// TIA Portal project "2022.11.22_双轴仿真2" (V17)
// Vorlageprojekt für das Buch mit Zielsystem S7-1200

(* hardware
DEVICE "S7-1200-Station_1"  S7-1200 Station
   slot 0: "Baugruppenträger_0"  Rack  V1.0
   slot 1: "PLC_1"  CPU 1214C DC/DC/DC  6ES7 214-1AG40-0XB0  V4.5
*)

// ===== PLC "PLC_1"  CPU 1214C DC/DC/DC =====

VAR_GLOBAL   // PLC tag table "Standard-Variablentabelle"
   "感应器5" AT %I1.1 : Bool;
   "感应器6" AT %I1.2 : Bool;
   "输入预留3" AT %I1.3 : Bool;
   "输入预留4" AT %I1.4 : Bool;
   "输入预留5" AT %I1.5 : Bool;
   "输入预留6" AT %I1.6 : Bool;
   "输入预留7" AT %I1.7 : Bool;
   "传送带4" AT %Q0.3 : Bool;
   "输出预留2" AT %Q0.7 : Bool;
   "输出预留3" AT %Q1.2 : Bool;
   "输出预留4" AT %Q1.5 : Bool;
   "输出预留5" AT %Q1.6 : Bool;
   "输出预留6" AT %Q1.7 : Bool;
   "启动" AT %M10.0 : Bool;
   "物体1执行步" AT %MD400 : DWord;
   "物体2执行步" AT %MD404 : DWord;
   "物体3执行步" AT %MD408 : DWord;
   "上升沿" AT %M100.0 : Bool;
   "上升沿(1)" AT %M100.1 : Bool;
   "上升沿(2)" AT %M100.2 : Bool;
END_VAR

VAR_GLOBAL   // PLC tag table "XML 中的变量表_1"
   "感应器1" AT %I0.0 : Bool;
   "感应器2" AT %I0.1 : Bool;
   "感应器3" AT %I0.2 : Bool;
   "感应器4" AT %I0.3 : Bool;
   "X动作感应" AT %I0.4 : Bool;
   "Z动作感应" AT %I0.5 : Bool;
   "吸物旋转到位" AT %I0.6 : Bool;
   "旋转到位" AT %I0.7 : Bool;
   "有物感应" AT %I1.0 : Bool;
   "传送带1" AT %Q0.0 : Bool;
   "传送带2" AT %Q0.1 : Bool;
   "传送带3" AT %Q0.2 : Bool;
   "X气缸" AT %Q0.4 : Bool;
   "Z气缸" AT %Q0.5 : Bool;
   "吸物" AT %Q0.6 : Bool;
   "顺时针90度" AT %Q1.0 : Bool;
   "逆时针90度" AT %Q1.1 : Bool;
   "吸物顺时针旋转" AT %Q1.3 : Bool;
   "吸物逆时针旋转" AT %Q1.4 : Bool;
END_VAR

DATA_BLOCK "数据块_1"   // DB1
{ S7_Optimized_Access := 'TRUE' }
VERSION : 0.1
   VAR
      计时器 : Array[0..100] of IEC_TIMER;
   END_VAR
BEGIN
END_DATA_BLOCK

FUNCTION "物体1" : Void   // FC1, LAD
{ S7_Optimized_Access := 'TRUE' }
VERSION : 0.1
   VAR_TEMP   // added for the SCL form of the ladder/FBD networks
      _w1 : Bool;
      _w2 : Bool;
   END_VAR
BEGIN

REGION Network 1: 30 伸出X气缸
   // 传输30个数据后  X气缸置位 运行   并同时传输数据40个数据  1执行步
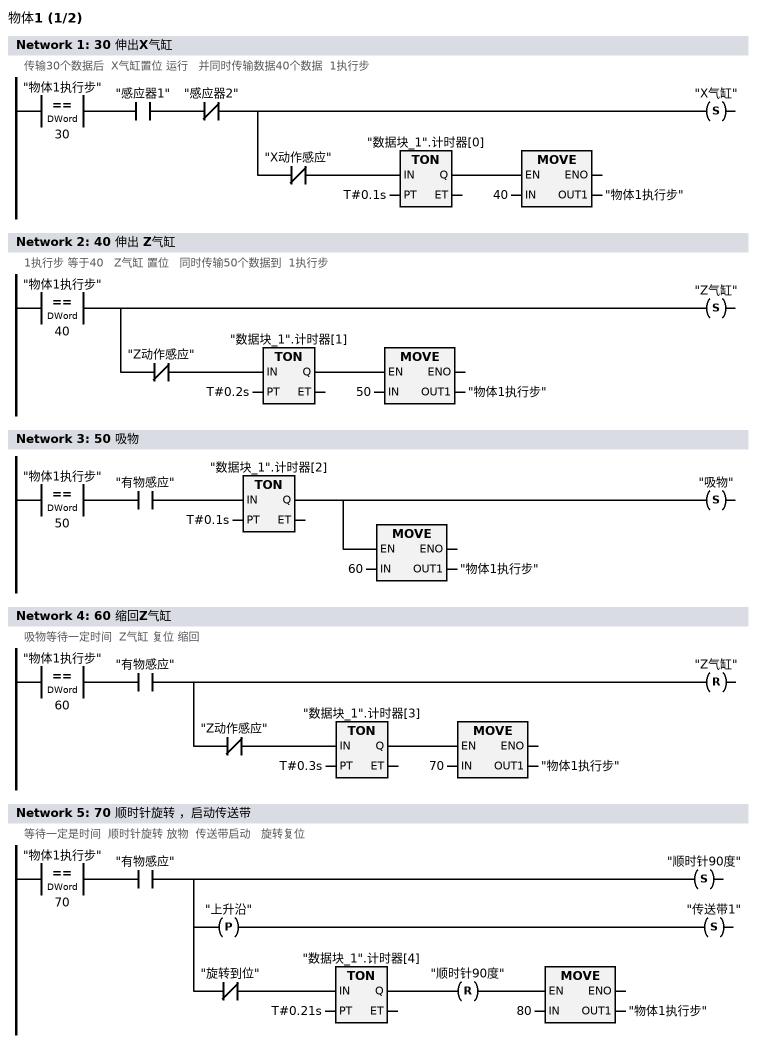
   #_w1 := ("物体1执行步" = 30) AND "感应器1" AND NOT "感应器2";
   IF #_w1 THEN "X气缸" := TRUE; END_IF;
   "数据块_1".计时器[0].TON(IN := #_w1 AND NOT "X动作感应", PT := T#0.1s);
   IF "数据块_1".计时器[0].Q THEN "物体1执行步" := 40; END_IF;
END_REGION

REGION Network 2: 40 伸出 Z气缸
   // 1执行步 等于40   Z气缸 置位   同时传输50个数据到  1执行步
   #_w1 := "物体1执行步" = 40;
   IF #_w1 THEN "Z气缸" := TRUE; END_IF;
   "数据块_1".计时器[1].TON(IN := #_w1 AND NOT "Z动作感应", PT := T#0.2s);
   IF "数据块_1".计时器[1].Q THEN "物体1执行步" := 50; END_IF;
END_REGION

REGION Network 3: 50 吸物
   "数据块_1".计时器[2].TON(IN := ("物体1执行步" = 50) AND "有物感应", PT := T#0.1s);
   IF "数据块_1".计时器[2].Q THEN
       "吸物" := TRUE;
       "物体1执行步" := 60;
   END_IF;
END_REGION

REGION Network 4: 60 缩回Z气缸
   // 吸物等待一定时间  Z气缸 复位 缩回
   #_w1 := ("物体1执行步" = 60) AND "有物感应";
   IF #_w1 THEN "Z气缸" := FALSE; END_IF;
   "数据块_1".计时器[3].TON(IN := #_w1 AND NOT "Z动作感应", PT := T#0.3s);
   IF "数据块_1".计时器[3].Q THEN "物体1执行步" := 70; END_IF;
END_REGION

REGION Network 5: 70 顺时针旋转 ，启动传送带
   // 等待一定是时间  顺时针旋转 放物  传送带启动   旋转复位
   #_w1 := ("物体1执行步" = 70) AND "有物感应";
   IF #_w1 THEN "顺时针90度" := TRUE; END_IF;
   #_w2 := #_w1 AND NOT "上升沿";   // rising edge
   "上升沿" := #_w1;
   IF #_w2 THEN "传送带1" := TRUE; END_IF;
   "数据块_1".计时器[4].TON(IN := #_w1 AND NOT "旋转到位", PT := T#0.21s);
   IF "数据块_1".计时器[4].Q THEN
       "顺时针90度" := FALSE;
       "物体1执行步" := 80;
   END_IF;
END_REGION

REGION Network 6: 80 伸出 Z气缸 停止传送2
   // 旋转放物  传送带2停止
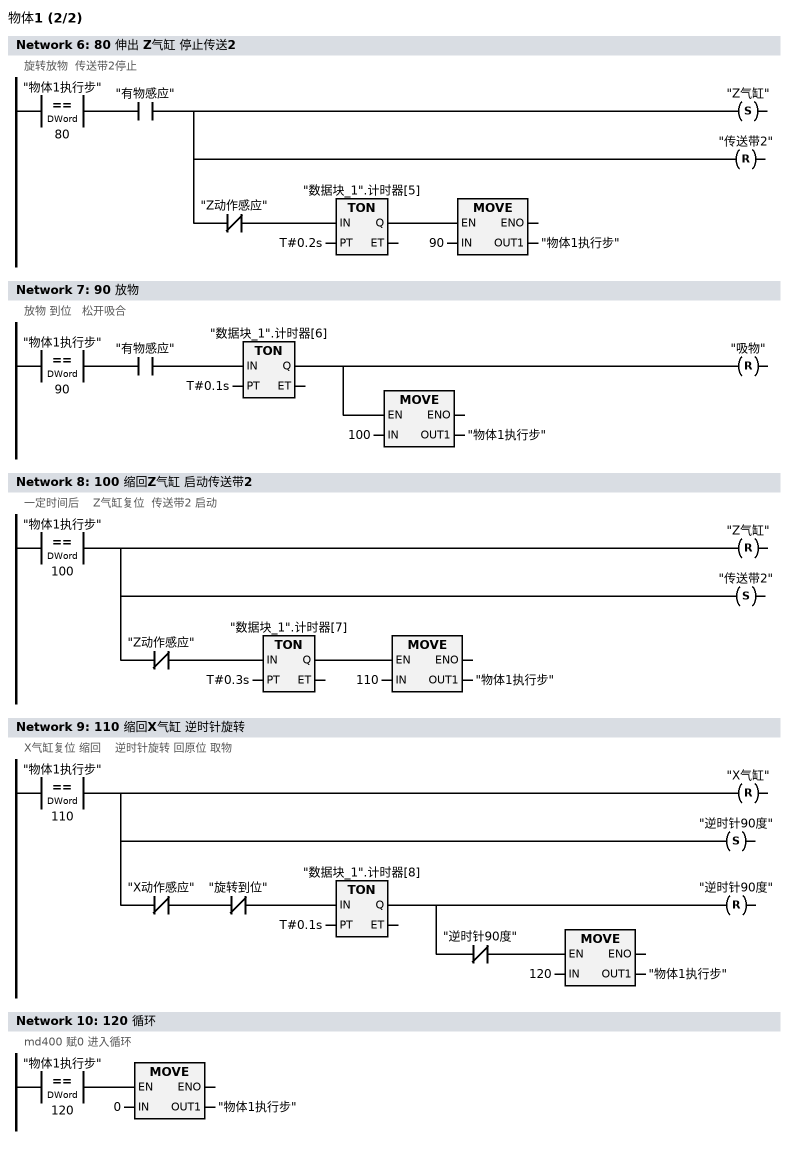
   #_w1 := ("物体1执行步" = 80) AND "有物感应";
   IF #_w1 THEN
       "Z气缸" := TRUE;
       "传送带2" := FALSE;
   END_IF;
   "数据块_1".计时器[5].TON(IN := #_w1 AND NOT "Z动作感应", PT := T#0.2s);
   IF "数据块_1".计时器[5].Q THEN "物体1执行步" := 90; END_IF;
END_REGION

REGION Network 7: 90 放物
   // 放物 到位   松开吸合
   "数据块_1".计时器[6].TON(IN := ("物体1执行步" = 90) AND "有物感应", PT := T#0.1s);
   IF "数据块_1".计时器[6].Q THEN
       "吸物" := FALSE;
       "物体1执行步" := 100;
   END_IF;
END_REGION

REGION Network 8: 100 缩回Z气缸 启动传送带2
   // 一定时间后    Z气缸复位  传送带2 启动
   #_w1 := "物体1执行步" = 100;
   IF #_w1 THEN
       "Z气缸" := FALSE;
       "传送带2" := TRUE;
   END_IF;
   "数据块_1".计时器[7].TON(IN := #_w1 AND NOT "Z动作感应", PT := T#0.3s);
   IF "数据块_1".计时器[7].Q THEN "物体1执行步" := 110; END_IF;
END_REGION

REGION Network 9: 110 缩回X气缸 逆时针旋转
   // X气缸复位 缩回    逆时针旋转 回原位 取物
   #_w1 := "物体1执行步" = 110;
   IF #_w1 THEN
       "X气缸" := FALSE;
       "逆时针90度" := TRUE;
   END_IF;
   "数据块_1".计时器[8].TON(IN := #_w1 AND NOT "X动作感应" AND NOT "旋转到位", PT := T#0.1s);
   IF "数据块_1".计时器[8].Q THEN "逆时针90度" := FALSE; END_IF;
   IF "数据块_1".计时器[8].Q AND NOT "逆时针90度" THEN "物体1执行步" := 120; END_IF;
END_REGION

REGION Network 10: 120 循环
   // md400 赋0 进入循环
   RUNG wire#powerrail
      { S7_Templates := "SrcType := DWord" } EQ_Contact(in1 := "物体1执行步", in2 := 120)
      Move(in := 0, out1 => "物体1执行步")
   END_RUNG
   // the same network as SCL:
   IF "物体1执行步" = 120 THEN "物体1执行步" := 0; END_IF;
END_REGION
END_FUNCTION

FUNCTION "物体2" : Void   // FC2, LAD
{ S7_Optimized_Access := 'TRUE' }
VERSION : 0.1
   VAR_TEMP   // added for the SCL form of the ladder/FBD networks
      _w1 : Bool;
      _w2 : Bool;
   END_VAR
BEGIN

REGION Network 1: 360 伸出 X气缸
   // 感应传感器 1 2 同时工作
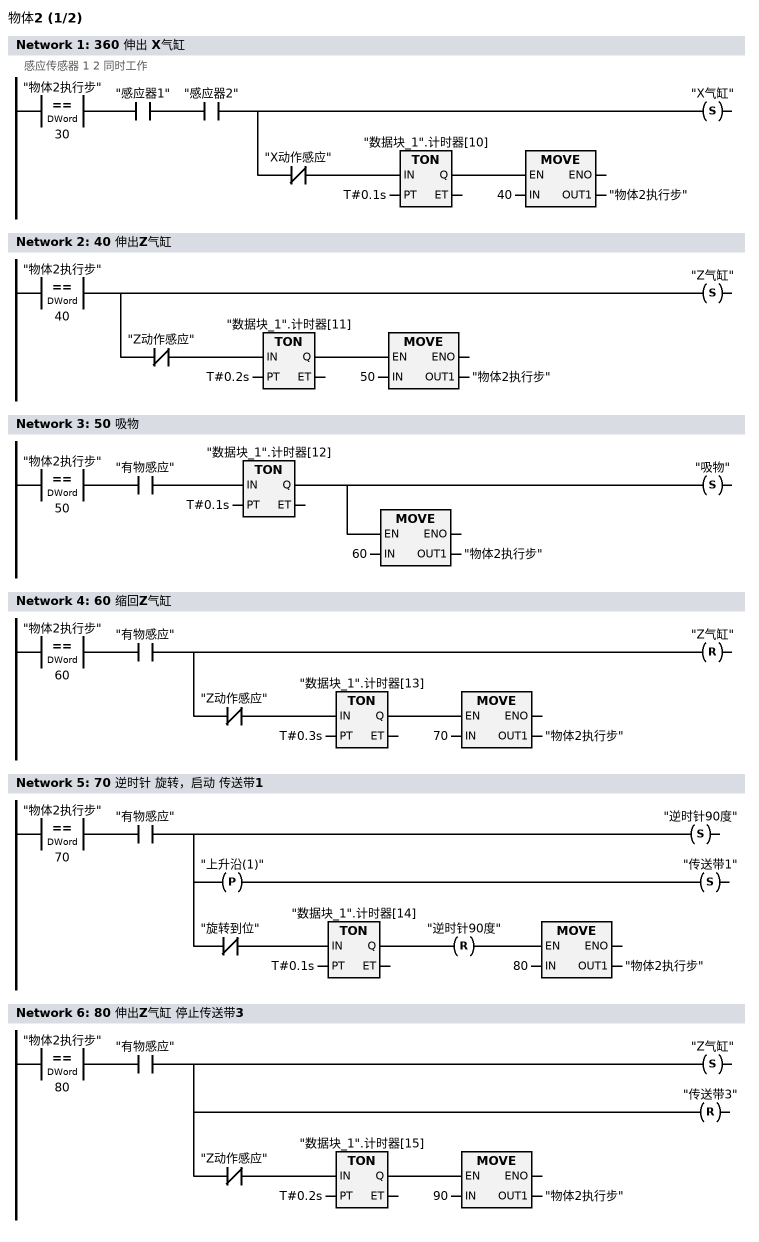
   #_w1 := ("物体2执行步" = 30) AND "感应器1" AND "感应器2";
   IF #_w1 THEN "X气缸" := TRUE; END_IF;
   "数据块_1".计时器[10].TON(IN := #_w1 AND NOT "X动作感应", PT := T#0.1s);
   IF "数据块_1".计时器[10].Q THEN "物体2执行步" := 40; END_IF;
END_REGION

REGION Network 2: 40 伸出Z气缸
   #_w1 := "物体2执行步" = 40;
   IF #_w1 THEN "Z气缸" := TRUE; END_IF;
   "数据块_1".计时器[11].TON(IN := #_w1 AND NOT "Z动作感应", PT := T#0.2s);
   IF "数据块_1".计时器[11].Q THEN "物体2执行步" := 50; END_IF;
END_REGION

REGION Network 3: 50 吸物
   "数据块_1".计时器[12].TON(IN := ("物体2执行步" = 50) AND "有物感应", PT := T#0.1s);
   IF "数据块_1".计时器[12].Q THEN
       "吸物" := TRUE;
       "物体2执行步" := 60;
   END_IF;
END_REGION

REGION Network 4: 60 缩回Z气缸
   #_w1 := ("物体2执行步" = 60) AND "有物感应";
   IF #_w1 THEN "Z气缸" := FALSE; END_IF;
   "数据块_1".计时器[13].TON(IN := #_w1 AND NOT "Z动作感应", PT := T#0.3s);
   IF "数据块_1".计时器[13].Q THEN "物体2执行步" := 70; END_IF;
END_REGION

REGION Network 5: 70 逆时针 旋转，启动 传送带1
   #_w1 := ("物体2执行步" = 70) AND "有物感应";
   IF #_w1 THEN "逆时针90度" := TRUE; END_IF;
   #_w2 := #_w1 AND NOT "上升沿(1)";   // rising edge
   "上升沿(1)" := #_w1;
   IF #_w2 THEN "传送带1" := TRUE; END_IF;
   "数据块_1".计时器[14].TON(IN := #_w1 AND NOT "旋转到位", PT := T#0.1s);
   IF "数据块_1".计时器[14].Q THEN
       "逆时针90度" := FALSE;
       "物体2执行步" := 80;
   END_IF;
END_REGION

REGION Network 6: 80 伸出Z气缸 停止传送带3
   #_w1 := ("物体2执行步" = 80) AND "有物感应";
   IF #_w1 THEN
       "Z气缸" := TRUE;
       "传送带3" := FALSE;
   END_IF;
   "数据块_1".计时器[15].TON(IN := #_w1 AND NOT "Z动作感应", PT := T#0.2s);
   IF "数据块_1".计时器[15].Q THEN "物体2执行步" := 90; END_IF;
END_REGION

REGION Network 7: 90 放物
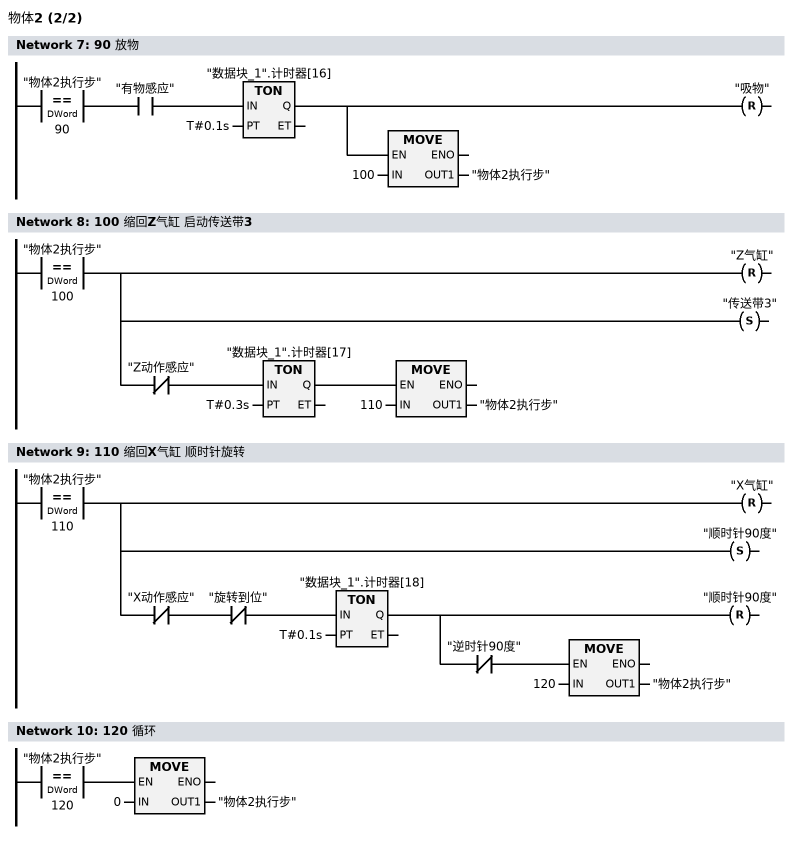
   "数据块_1".计时器[16].TON(IN := ("物体2执行步" = 90) AND "有物感应", PT := T#0.1s);
   IF "数据块_1".计时器[16].Q THEN
       "吸物" := FALSE;
       "物体2执行步" := 100;
   END_IF;
END_REGION

REGION Network 8: 100 缩回Z气缸 启动传送带3
   #_w1 := "物体2执行步" = 100;
   IF #_w1 THEN
       "Z气缸" := FALSE;
       "传送带3" := TRUE;
   END_IF;
   "数据块_1".计时器[17].TON(IN := #_w1 AND NOT "Z动作感应", PT := T#0.3s);
   IF "数据块_1".计时器[17].Q THEN "物体2执行步" := 110; END_IF;
END_REGION

REGION Network 9: 110 缩回X气缸 顺时针旋转
   #_w1 := "物体2执行步" = 110;
   IF #_w1 THEN
       "X气缸" := FALSE;
       "顺时针90度" := TRUE;
   END_IF;
   "数据块_1".计时器[18].TON(IN := #_w1 AND NOT "X动作感应" AND NOT "旋转到位", PT := T#0.1s);
   IF "数据块_1".计时器[18].Q THEN "顺时针90度" := FALSE; END_IF;
   IF "数据块_1".计时器[18].Q AND NOT "逆时针90度" THEN "物体2执行步" := 120; END_IF;
END_REGION

REGION Network 10: 120 循环
   RUNG wire#powerrail
      { S7_Templates := "SrcType := DWord" } EQ_Contact(in1 := "物体2执行步", in2 := 120)
      Move(in := 0, out1 => "物体2执行步")
   END_RUNG
   // the same network as SCL:
   IF "物体2执行步" = 120 THEN "物体2执行步" := 0; END_IF;
END_REGION
END_FUNCTION

FUNCTION "物体3" : Void   // FC3, LAD
{ S7_Optimized_Access := 'TRUE' }
VERSION : 0.1
   VAR_TEMP   // added for the SCL form of the ladder/FBD networks
      _w1 : Bool;
      _w2 : Bool;
   END_VAR
BEGIN

REGION Network 1: 360 伸出 X气缸
   // 感应传感器 1 2 同时工作
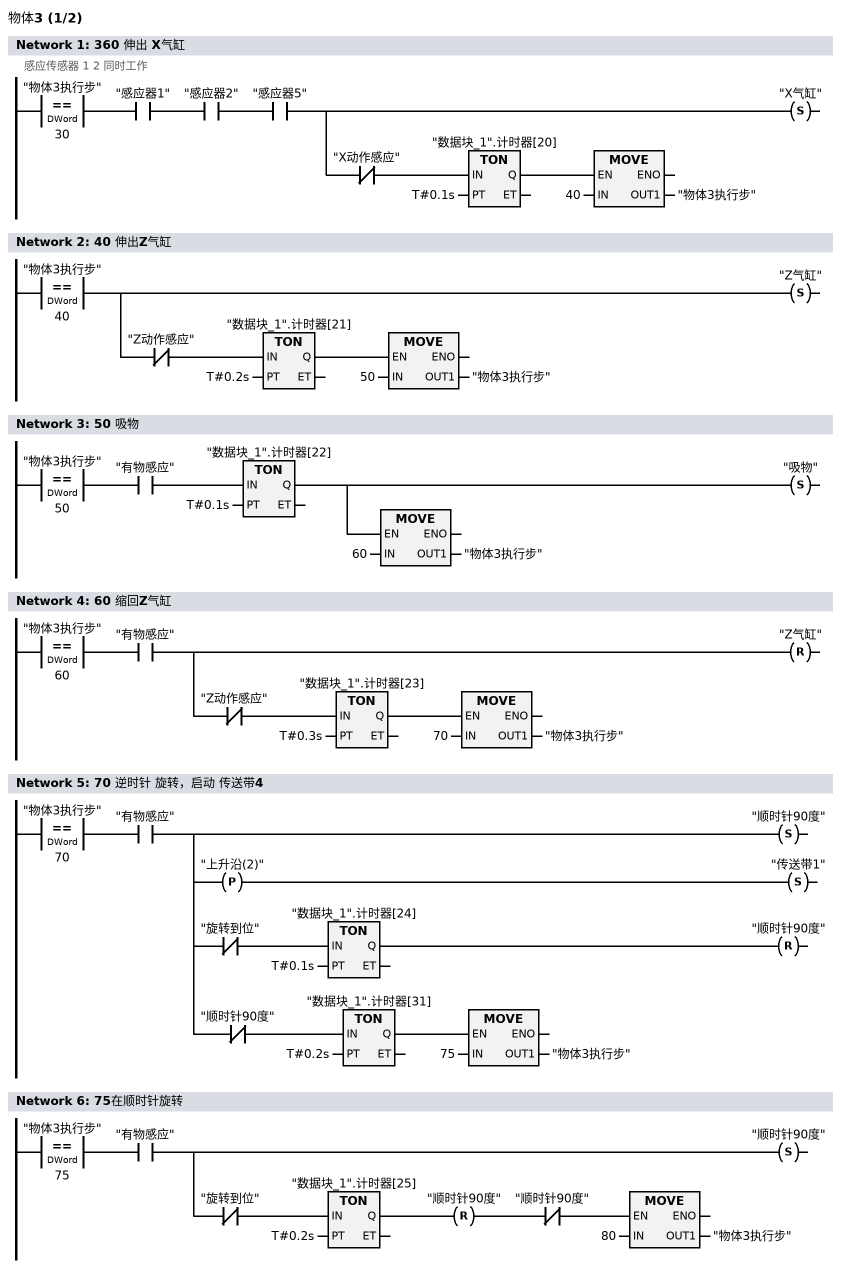
   #_w1 := ("物体3执行步" = 30) AND "感应器1" AND "感应器2" AND "感应器5";
   IF #_w1 THEN "X气缸" := TRUE; END_IF;
   "数据块_1".计时器[20].TON(IN := #_w1 AND NOT "X动作感应", PT := T#0.1s);
   IF "数据块_1".计时器[20].Q THEN "物体3执行步" := 40; END_IF;
END_REGION

REGION Network 2: 40 伸出Z气缸
   #_w1 := "物体3执行步" = 40;
   IF #_w1 THEN "Z气缸" := TRUE; END_IF;
   "数据块_1".计时器[21].TON(IN := #_w1 AND NOT "Z动作感应", PT := T#0.2s);
   IF "数据块_1".计时器[21].Q THEN "物体3执行步" := 50; END_IF;
END_REGION

REGION Network 3: 50 吸物
   "数据块_1".计时器[22].TON(IN := ("物体3执行步" = 50) AND "有物感应", PT := T#0.1s);
   IF "数据块_1".计时器[22].Q THEN
       "吸物" := TRUE;
       "物体3执行步" := 60;
   END_IF;
END_REGION

REGION Network 4: 60 缩回Z气缸
   #_w1 := ("物体3执行步" = 60) AND "有物感应";
   IF #_w1 THEN "Z气缸" := FALSE; END_IF;
   "数据块_1".计时器[23].TON(IN := #_w1 AND NOT "Z动作感应", PT := T#0.3s);
   IF "数据块_1".计时器[23].Q THEN "物体3执行步" := 70; END_IF;
END_REGION

REGION Network 5: 70 逆时针 旋转，启动 传送带4
   #_w1 := ("物体3执行步" = 70) AND "有物感应";
   IF #_w1 THEN "顺时针90度" := TRUE; END_IF;
   #_w2 := #_w1 AND NOT "上升沿(2)";   // rising edge
   "上升沿(2)" := #_w1;
   IF #_w2 THEN "传送带1" := TRUE; END_IF;
   "数据块_1".计时器[24].TON(IN := #_w1 AND NOT "旋转到位", PT := T#0.1s);
   IF "数据块_1".计时器[24].Q THEN "顺时针90度" := FALSE; END_IF;
   "数据块_1".计时器[31].TON(IN := #_w1 AND NOT "顺时针90度", PT := T#0.2s);
   IF "数据块_1".计时器[31].Q THEN "物体3执行步" := 75; END_IF;
END_REGION

REGION Network 6: 75在顺时针旋转
   #_w1 := ("物体3执行步" = 75) AND "有物感应";
   IF #_w1 THEN "顺时针90度" := TRUE; END_IF;
   "数据块_1".计时器[25].TON(IN := #_w1 AND NOT "旋转到位", PT := T#0.2s);
   IF "数据块_1".计时器[25].Q THEN "顺时针90度" := FALSE; END_IF;
   IF "数据块_1".计时器[25].Q AND NOT "顺时针90度" THEN "物体3执行步" := 80; END_IF;
END_REGION

REGION Network 7: 80 伸出Z气缸 停止传送带4
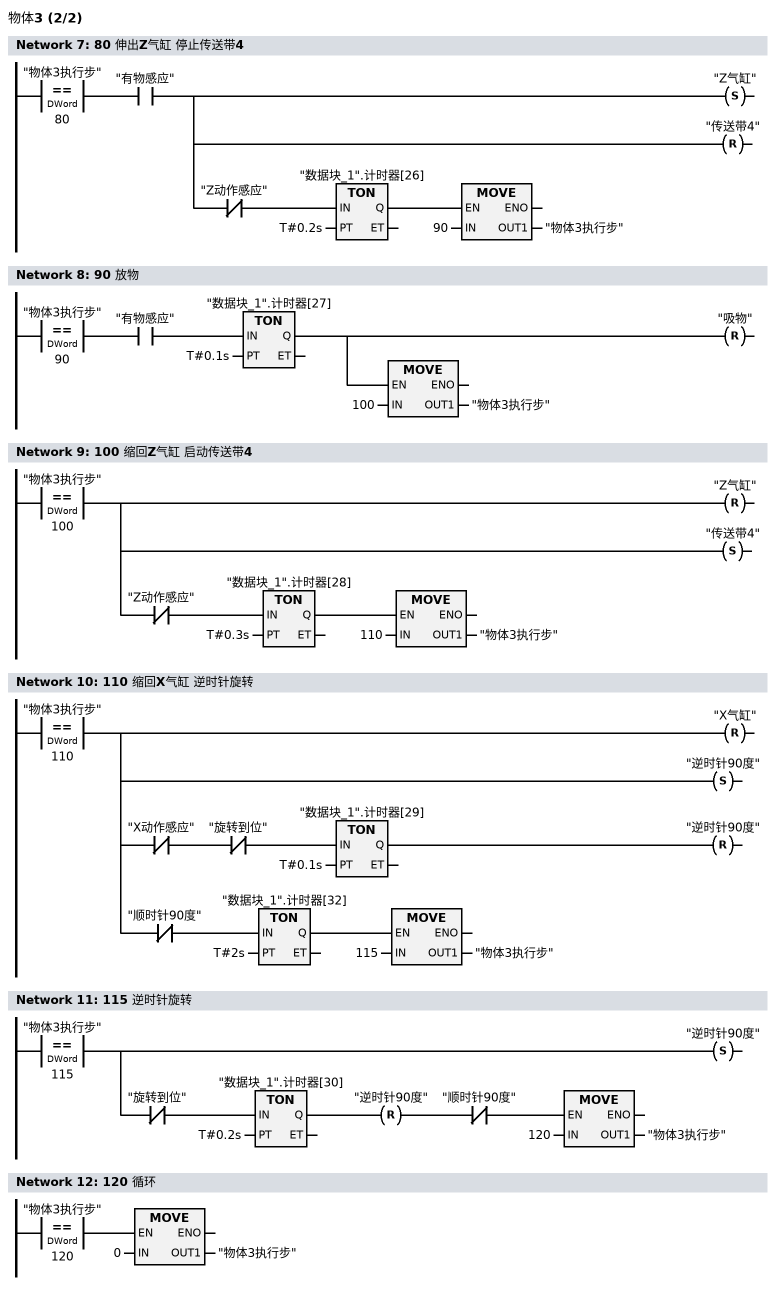
   #_w1 := ("物体3执行步" = 80) AND "有物感应";
   IF #_w1 THEN
       "Z气缸" := TRUE;
       "传送带4" := FALSE;
   END_IF;
   "数据块_1".计时器[26].TON(IN := #_w1 AND NOT "Z动作感应", PT := T#0.2s);
   IF "数据块_1".计时器[26].Q THEN "物体3执行步" := 90; END_IF;
END_REGION

REGION Network 8: 90 放物
   "数据块_1".计时器[27].TON(IN := ("物体3执行步" = 90) AND "有物感应", PT := T#0.1s);
   IF "数据块_1".计时器[27].Q THEN
       "吸物" := FALSE;
       "物体3执行步" := 100;
   END_IF;
END_REGION

REGION Network 9: 100 缩回Z气缸 启动传送带4
   #_w1 := "物体3执行步" = 100;
   IF #_w1 THEN
       "Z气缸" := FALSE;
       "传送带4" := TRUE;
   END_IF;
   "数据块_1".计时器[28].TON(IN := #_w1 AND NOT "Z动作感应", PT := T#0.3s);
   IF "数据块_1".计时器[28].Q THEN "物体3执行步" := 110; END_IF;
END_REGION

REGION Network 10: 110 缩回X气缸 逆时针旋转
   #_w1 := "物体3执行步" = 110;
   IF #_w1 THEN
       "X气缸" := FALSE;
       "逆时针90度" := TRUE;
   END_IF;
   "数据块_1".计时器[29].TON(IN := #_w1 AND NOT "X动作感应" AND NOT "旋转到位", PT := T#0.1s);
   IF "数据块_1".计时器[29].Q THEN "逆时针90度" := FALSE; END_IF;
   "数据块_1".计时器[32].TON(IN := #_w1 AND NOT "顺时针90度", PT := T#2s);
   IF "数据块_1".计时器[32].Q THEN "物体3执行步" := 115; END_IF;
END_REGION

REGION Network 11: 115 逆时针旋转
   #_w1 := "物体3执行步" = 115;
   IF #_w1 THEN "逆时针90度" := TRUE; END_IF;
   "数据块_1".计时器[30].TON(IN := #_w1 AND NOT "旋转到位", PT := T#0.2s);
   IF "数据块_1".计时器[30].Q THEN "逆时针90度" := FALSE; END_IF;
   IF "数据块_1".计时器[30].Q AND NOT "顺时针90度" THEN "物体3执行步" := 120; END_IF;
END_REGION

REGION Network 12: 120 循环
   RUNG wire#powerrail
      { S7_Templates := "SrcType := DWord" } EQ_Contact(in1 := "物体3执行步", in2 := 120)
      Move(in := 0, out1 => "物体3执行步")
   END_RUNG
   // the same network as SCL:
   IF "物体3执行步" = 120 THEN "物体3执行步" := 0; END_IF;
END_REGION
END_FUNCTION

FUNCTION "MHJ-PLC-Lab-Function-S71200" : Void   // FC9000, SCL
{ S7_Optimized_Access := 'TRUE' }
VERSION : 0.1
   VAR_TEMP
      rdTimeReturn : Int;
      outputTime : DTL;
      SyncVal : Byte;
      forVal : Int;
      forVal_2 : Int;
      Value : Byte;
   END_VAR
   VAR CONSTANT
      CompVal : Byte := 16#34;
      Value_01 : Byte := 16#11;
      Value_01_DW : DWord := 16#A165_D992;
      Value_02_DW : DWord := 16#58BE_4401;
   END_VAR
BEGIN

   #Value:=PEEK(area := 16#82,
        dbNumber := 0,
        byteOffset := 511);
   #Value := #Value + 1;

   POKE(area := 16#82,
        dbNumber := 0,
        byteOffset := 511,
        value := #Value);

   POKE(area:=16#81,
        dbNumber:=0,
        byteOffset:=1016,
        value:=#Value_01_DW);
   POKE(area := 16#81,
        dbNumber := 0,
        byteOffset := 1020,
        value := #Value_02_DW);

   POKE(area := 16#81,
        dbNumber := 0,
        byteOffset := 511,
        value := B#16#00);

   FOR #forVal := 0 TO 120 DO
       FOR #forVal_2:=0 TO 10 DO
           #rdTimeReturn:=RD_SYS_T(#outputTime);
           #rdTimeReturn := WR_SYS_T(#outputTime);
           #rdTimeReturn := RD_SYS_T(#outputTime);
           #rdTimeReturn := WR_SYS_T(#outputTime);
       END_FOR;
       #SyncVal:= PEEK(area := 16#81,
                      dbNumber := 0,
                      byteOffset := 511);
       IF #SyncVal = #CompVal THEN
          GOTO M_1;
       END_IF;
   END_FOR;
   RETURN;

   M_1:
   POKE(area := 16#81,
        dbNumber := 0,
        byteOffset := 511,
        value := B#16#0);
END_FUNCTION

ORGANIZATION_BLOCK "Main"   // OB1, LAD, ProgramCycle
TITLE = "Main Program Sweep (Cycle)"
{ S7_Optimized_Access := 'TRUE' }
VERSION : 0.1
   VAR_INPUT
      Initial_Call : Bool;   // Initial call of this OB
      Remanence : Bool;   // =True, if remanent data are available
   END_VAR
   VAR_TEMP   // added for the SCL form of the ladder/FBD networks
      _w1 : Bool;
      _w2 : Bool;
   END_VAR
BEGIN

REGION Network 1
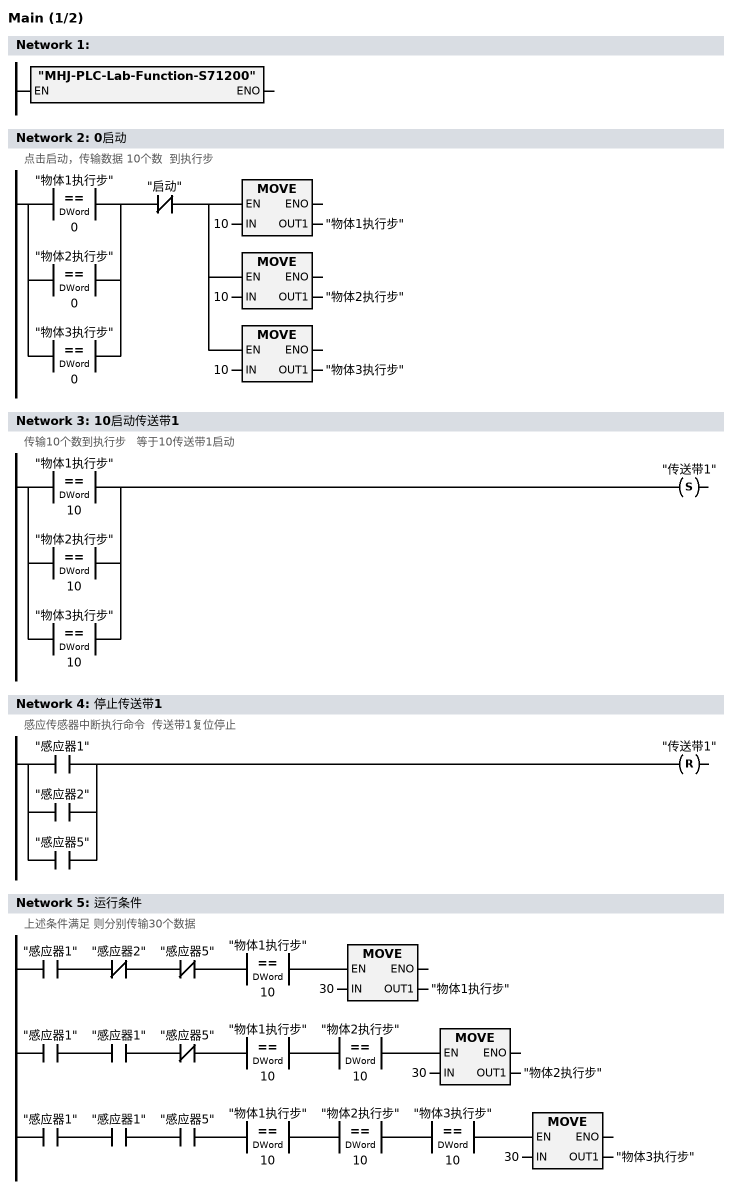
   RUNG wire#powerrail
      "MHJ-PLC-Lab-Function-S71200"()
   END_RUNG
   // the same network as SCL:
   "MHJ-PLC-Lab-Function-S71200"();
END_REGION

REGION Network 2: 0启动
   // 点击启动，传输数据 10个数  到执行步
   RUNG wire#powerrail
      { S7_Templates := "SrcType := DWord" } EQ_Contact(in1 := "物体1执行步", in2 := 0)
      wire#w1
      I_Contact( "启动" )
      wire#w2
      Move(in := 10, out1 => "物体1执行步")
   END_RUNG
   RUNG wire#powerrail
      { S7_Templates := "SrcType := DWord" } EQ_Contact(in1 := "物体2执行步", in2 := 0)
   END_RUNG wire#w1
   RUNG wire#powerrail
      { S7_Templates := "SrcType := DWord" } EQ_Contact(in1 := "物体3执行步", in2 := 0)
   END_RUNG wire#w1
   RUNG wire#w2
      Move(in := 10, out1 => "物体2执行步")
   END_RUNG
   RUNG wire#w2
      Move(in := 10, out1 => "物体3执行步")
   END_RUNG
   // the same network as SCL:
   #_w1 := (("物体1执行步" = 0) OR ("物体2执行步" = 0) OR ("物体3执行步" = 0)) AND NOT "启动";
   IF #_w1 THEN
       "物体1执行步" := 10;
       "物体2执行步" := 10;
       "物体3执行步" := 10;
   END_IF;
END_REGION

REGION Network 3: 10启动传送带1
   // 传输10个数到执行步   等于10传送带1启动
   RUNG wire#powerrail
      { S7_Templates := "SrcType := DWord" } EQ_Contact(in1 := "物体1执行步", in2 := 10)
      wire#w1
      S_Coil( "传送带1" )
   END_RUNG
   RUNG wire#powerrail
      { S7_Templates := "SrcType := DWord" } EQ_Contact(in1 := "物体2执行步", in2 := 10)
   END_RUNG wire#w1
   RUNG wire#powerrail
      { S7_Templates := "SrcType := DWord" } EQ_Contact(in1 := "物体3执行步", in2 := 10)
   END_RUNG wire#w1
   // the same network as SCL:
   IF ("物体1执行步" = 10) OR ("物体2执行步" = 10) OR ("物体3执行步" = 10) THEN "传送带1" := TRUE; END_IF;
END_REGION

REGION Network 4: 停止传送带1
   // 感应传感器中断执行命令  传送带1复位停止
   RUNG wire#powerrail
      Contact( "感应器1" )
      wire#w1
      R_Coil( "传送带1" )
   END_RUNG
   RUNG wire#powerrail
      Contact( "感应器2" )
   END_RUNG wire#w1
   RUNG wire#powerrail
      Contact( "感应器5" )
   END_RUNG wire#w1
   // the same network as SCL:
   IF "感应器1" OR "感应器2" OR "感应器5" THEN "传送带1" := FALSE; END_IF;
END_REGION

REGION Network 5: 运行条件
   // 上述条件满足 则分别传输30个数据
   RUNG wire#powerrail
      Contact( "感应器1" )
      I_Contact( "感应器2" )
      I_Contact( "感应器5" )
      { S7_Templates := "SrcType := DWord" } EQ_Contact(in1 := "物体1执行步", in2 := 10)
      Move(in := 30, out1 => "物体1执行步")
   END_RUNG
   RUNG wire#powerrail
      Contact( "感应器1" )
      Contact( "感应器1" )
      I_Contact( "感应器5" )
      { S7_Templates := "SrcType := DWord" } EQ_Contact(in1 := "物体1执行步", in2 := 10)
      { S7_Templates := "SrcType := DWord" } EQ_Contact(in1 := "物体2执行步", in2 := 10)
      Move(in := 30, out1 => "物体2执行步")
   END_RUNG
   RUNG wire#powerrail
      Contact( "感应器1" )
      Contact( "感应器1" )
      Contact( "感应器5" )
      { S7_Templates := "SrcType := DWord" } EQ_Contact(in1 := "物体1执行步", in2 := 10)
      { S7_Templates := "SrcType := DWord" } EQ_Contact(in1 := "物体2执行步", in2 := 10)
      { S7_Templates := "SrcType := DWord" } EQ_Contact(in1 := "物体3执行步", in2 := 10)
      Move(in := 30, out1 => "物体3执行步")
   END_RUNG
   // the same network as SCL:
   IF "感应器1" AND NOT "感应器2" AND NOT "感应器5" AND ("物体1执行步" = 10) THEN "物体1执行步" := 30; END_IF;
   IF "感应器1" AND "感应器1" AND NOT "感应器5" AND ("物体1执行步" = 10) AND ("物体2执行步" = 10) THEN "物体2执行步" := 30; END_IF;
   IF "感应器1" AND "感应器1" AND "感应器5" AND ("物体1执行步" = 10) AND ("物体2执行步" = 10) AND ("物体3执行步" = 10) THEN
       "物体3执行步" := 30;
   END_IF;
END_REGION

REGION Network 6
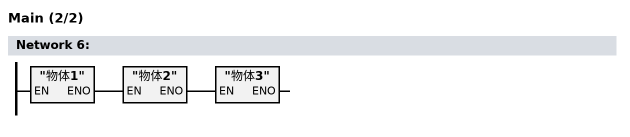
   RUNG wire#powerrail
      "物体1"()
      "物体2"()
      "物体3"()
   END_RUNG
   // the same network as SCL:
   "物体1"(ENO => #_w1);
   "物体2"(EN := #_w1, ENO => #_w2);
   IF #_w2 THEN "物体3"(); END_IF;
END_REGION
END_ORGANIZATION_BLOCK